PROGRAM POU
VAR
END_VAR

END_PROGRAM

(* stored: Version 1.1.0.1, ProductVersion 3.1.4022.12
   POU POU: Id {df32000e-33bd-42ab-8dd0-7c1ad55e1bfd}, SpecialFunc None *)
